GLOBALCONSTANTS AID_LA (* Line attributes object attribute ids *)
  (* Standard: 61499-1; Description: Copyright (c) 2023 HR Agrartechnik GmbH This program and the accompanying materials are made available under the terms of the Eclipse Public License 2.0 which is available at https://www.eclipse.org/legal/epl-2.0/ SPDX-License-Identifier: EPL-2.0 *)
  (* Version 1.0, 2026-06-20, Franz Höpfinger, HR Agrartechnik GmbH *)
  PACKAGE isobus::UT::Q::const::AID;
  IMPORT eclipse4diac::core::TypeHash;
  VAR_GLOBAL CONSTANT
    LINE_COLOUR : USINT := USINT#1; (* 1: AID_LA_LINE_COLOUR *)
    LINE_WIDTH : USINT := USINT#2; (* 2: AID_LA_LINE_WIDTH *)
    LINE_ART : USINT := USINT#3; (* 3: AID_LA_LINE_ART - Bit pattern art for line (each bit represents a paintbrush spot). *)
  END_VAR
END_GLOBALCONSTANTS
